Yaskawa INFORM job: MASTER_X2.JBI

/JOB
//NAME MASTER_X2
///FOLDERNAME MASTER_ODWLOK
//POS
///NPOS 138,138,138,0,0,0
///TOOL 0
///POSTYPE PULSE
///PULSE
C00000=2000,-113621,-91819,0,89172,0
C00001=2000,-113621,-91819,0,89172,0
C00002=2000,-99612,-82443,0,53832,0
C00003=2000,-48025,-60869,0,102856,0
C00004=3643,-76224,-106676,19950,71810,76872
C00005=2000,-130321,-133031,0,28968,0
C00006=2000,-109649,-128472,0,44436,0
C00007=2000,-75195,-120874,0,70216,0
C00008=2000,-52226,-115808,0,87402,0
C00009=2000,-87067,-95572,0,78525,0
C00010=2000,-87067,-95572,0,78525,0
C00011=2000,-87067,-95572,0,78525,0
C00012=-12667,-135547,-130714,31270,45596,0
C00013=-12667,-135547,-130714,31270,45596,0
C00014=-12667,-135547,-130714,31270,45596,0
C00015=-7337,-135032,-132177,15524,30149,37578
C00016=-1415,-134459,-133802,-1969,12985,79332
C00017=-1415,-134459,-133802,-1969,12985,79332
C00018=-15972,-110889,-128286,-10965,59905,-43045
C00019=2800,-56338,-97337,-367,83074,232
C00020=2800,-56338,-97337,-367,83074,232
C00021=2000,-92772,-84335,0,66375,0
C00022=2000,-92772,-84335,0,66375,0
C00023=2000,-92772,-84335,0,66375,0
C00024=2000,-92772,-84335,0,66375,0
C00025=2000,-92055,-48789,0,51065,0
C00026=2000,-92055,-48789,0,51065,0
C00027=2000,-92055,-48789,0,51065,0
C00028=2000,-92055,-48789,0,51065,0
C00029=2348,-136985,-121477,16,96092,119
C00030=2348,-136985,-121477,16,96092,119
C00031=2348,-136985,-121477,16,96092,119
C00032=-9622,-119744,-117240,5707,89112,22022
C00033=-39612,-76551,-106625,19964,71626,76894
C00034=-8691,-94790,-119167,5108,91578,19600
C00035=1903,-101039,-123464,18,98414,-30
C00036=1903,-101039,-123464,18,98414,-30
C00037=1903,-101039,-123464,18,98414,-30
C00038=1903,-101039,-123464,18,98414,-30
C00039=-39612,-76551,-106625,19964,71626,76894
C00040=-39612,-76551,-106625,19964,71626,76894
C00041=-39612,-76551,-106625,19964,71626,76894
C00042=-39612,-76551,-106625,19964,71626,76894
C00043=-39612,-76551,-106625,19964,71626,76894
C00044=-39612,-76551,-106625,19964,71626,76894
C00045=-39612,-76551,-106625,19964,71626,76894
C00046=-39612,-76551,-106625,19964,71626,76894
C00047=-39612,-76551,-106625,19964,71626,76894
C00048=-10776,-116726,-133110,1428,79202,268
C00049=-10776,-116726,-133110,1428,79202,268
C00050=-10907,-117335,-90652,-18762,63715,-59495
C00051=-10907,-117335,-90652,-18762,63715,-59495
C00052=-10776,-116726,-133110,1428,79202,268
C00053=-10776,-116726,-133110,1428,79202,268
C00054=-10907,-117335,-90652,-18762,63715,-59495
C00055=2286,-107682,-96534,-81,71711,101
C00056=2286,-107682,-96534,-81,71711,101
C00057=2286,-107682,-96534,-81,71711,101
C00058=2000,-113393,-91320,0,88983,0
C00059=2000,-113393,-91320,0,88983,0
C00060=2000,-113393,-91320,0,88983,0
C00061=2000,-113393,-91320,0,88983,0
C00062=2000,-113393,-91320,0,88983,0
C00063=-39612,-76551,-106625,19964,71626,76894
C00064=-39612,-76551,-106625,19964,71626,76894
C00065=-39612,-76551,-106625,19964,71626,76894
C00066=-39612,-76551,-106625,19964,71626,76894
C00067=-39612,-76551,-106625,19964,71626,76894
C00068=-39612,-76551,-106625,19964,71626,76894
C00069=15474,202180,164610,0,0,38
C00070=15474,202180,164610,0,0,38
C00071=3643,-76224,-106676,19950,71810,76872
C00072=15474,202180,164610,0,0,38
C00073=15474,202180,164610,0,0,38
C00074=15474,202180,164610,0,0,38
C00075=3643,-76224,-106676,19950,71810,76872
C00076=3643,-61024,-22647,36971,32176,65178
C00077=15474,202180,164610,0,0,38
C00078=3643,-76224,-106676,19950,71810,76872
C00079=1588,-95931,-85547,-536,91020,-79
C00080=1588,-95931,-85547,-536,91020,-79
C00081=2000,-138093,-117084,0,0,0
C00082=3643,-76224,-106676,19950,71810,76872
C00083=2000,-138093,-117084,0,0,0
C00084=2000,-138093,-117084,0,0,0
C00085=1941,-102693,-129564,10,101994,-18
C00086=3643,-76224,-106676,19950,71810,76872
C00087=1074,-84890,-111921,820,92639,-133
C00088=1074,-84890,-111921,820,92639,-133
C00089=1999,-107637,-123410,0,80759,1
C00090=3643,-76224,-106676,19950,71810,76872
C00091=2000,17994,-60377,0,102988,0
C00092=2000,-95440,-72516,0,38121,0
C00093=1074,-84890,-111921,820,92639,-133
C00094=3643,-76224,-106676,19950,71810,76872
C00095=421,-73083,-90384,-286,80877,-488
C00096=421,-73083,-90384,-286,80877,-488
C00097=2000,-112988,-119327,0,83158,0
C00098=3643,-76224,-106676,19950,71810,76872
C00099=2000,-112988,-119327,0,83158,0
C00100=2000,-112988,-119327,0,83158,0
C00101=2000,-112988,-119327,0,83158,0
C00102=2000,-112988,-119327,0,83158,0
C00103=2082,-130750,-111396,-32,62200,31
C00104=3643,-76224,-106676,19950,71810,76872
C00105=2082,-130750,-111396,-32,62200,31
C00106=2082,-130750,-111396,-32,62200,31
C00107=1579,-114561,-88072,141,60969,-160
C00108=1579,-114561,-88072,141,60969,-160
C00109=1579,-114561,-88072,141,60969,-160
C00110=3643,-76224,-106676,19950,71810,76872
C00111=-137109,-187493,-133090,6705,82774,-76786
C00112=3643,-76224,-106676,19950,71810,76872
C00113=1579,-114561,-88072,141,60969,-160
C00114=1579,-114561,-88072,141,60969,-160
C00115=2000,-76909,-65168,0,90368,0
C00116=3643,-76224,-106676,19950,71810,76872
C00117=2000,-76909,-65168,0,90368,0
C00118=2000,-76909,-65168,0,90368,0
C00119=3322,-122452,-100913,-73,83322,449
C00120=3643,-76224,-106676,19950,71810,76872
C00121=3322,-122452,-100913,-73,83322,449
C00122=3322,-122452,-100913,-73,83322,449
C00123=3322,-122452,-100913,-73,83322,449
C00124=3322,-122452,-100913,-73,83322,449
C00125=3322,-122452,-100913,-73,83322,449
C00126=2822,-118876,-115474,-188,81202,276
C00127=2000,-115920,-83969,0,54247,0
C00128=2000,-115920,-83969,0,54247,0
C00129=3271,-119374,-120746,-350,28955,423
C00130=3271,-119374,-120746,-350,28955,423
C00131=3271,-119374,-120746,-350,28955,423
C00132=3271,-119374,-120746,-350,28955,423
C00133=3271,-119374,-120746,-350,28955,423
C00134=3270,-119374,-120745,-350,28960,423
C00135=3270,-119374,-120745,-350,28960,423
C00136=3271,-119374,-120746,-350,28955,423
C00137=2000,-113621,-91819,0,89172,0
BC00000=87189,671070,860070
BC00001=87189,689489,1075229
BC00002=0,666204,302418
BC00003=118464,666204,678996
BC00004=199464,674570,1075173
BC00005=200134,698532,1075229
BC00006=160320,689975,1054047
BC00007=93964,675713,1018743
BC00008=49726,666204,995208
BC00009=66580,674291,1075175
BC00010=66580,674291,1075175
BC00011=66580,674291,1075175
BC00012=78393,670967,1075175
BC00013=78393,670967,1075175
BC00014=78393,670967,1075175
BC00015=64389,679433,1075175
BC00016=48829,688840,1075175
BC00017=48829,688840,1075175
BC00018=21214,672831,1075175
BC00019=194082,666204,1075175
BC00020=194082,666204,1075175
BC00021=244954,666204,1064818
BC00022=244954,666204,1063150
BC00023=244954,666204,804590
BC00024=244954,666204,1062399
BC00025=198883,666204,1060496
BC00026=198883,666204,1063896
BC00027=198883,666204,632238
BC00028=198883,666204,632238
BC00029=133260,671337,1075175
BC00030=133260,671337,1075175
BC00031=133260,671337,1075175
BC00032=179494,672257,1075175
BC00033=295325,674563,1075175
BC00034=207960,671388,1071361
BC00035=178026,670300,1070054
BC00036=178026,670300,1070054
BC00037=178026,670300,1070054
BC00038=178026,670300,1070054
BC00039=295325,674563,1075175
BC00040=295325,674563,1075175
BC00041=295325,674563,1075175
BC00042=295325,674563,1075175
BC00043=295325,674563,1075175
BC00044=295325,674563,1075175
BC00045=295325,674563,1075175
BC00046=295325,674563,1075175
BC00047=295325,674563,1075175
BC00048=165820,667836,1075229
BC00049=165820,667836,1075229
BC00050=165820,667836,534036
BC00051=165820,667836,534036
BC00052=165820,667836,1075229
BC00053=165820,667836,1075229
BC00054=165820,667836,534036
BC00055=84306,671503,1075229
BC00056=84306,671503,1075229
BC00057=84306,671503,1075229
BC00058=87189,666204,1075229
BC00059=87189,666204,1075229
BC00060=87189,666204,1075229
BC00061=87189,666204,1075229
BC00062=87189,666204,1075229
BC00063=295325,674563,1075175
BC00064=295325,674563,1075175
BC00065=295325,674563,1075175
BC00066=295325,674563,1075175
BC00067=295325,674563,1075175
BC00068=295325,674563,1075175
BC00069=0,675528,1075229
BC00070=0,675528,1075229
BC00071=199464,674570,1075173
BC00072=0,675528,1075229
BC00073=0,675528,1075229
BC00074=0,675528,1075229
BC00075=199464,674570,1075173
BC00076=199464,674570,909039
BC00077=0,675528,1075229
BC00078=199464,674570,1075173
BC00079=197645,666204,680424
BC00080=197645,666204,680424
BC00081=166720,666220,1057063
BC00082=199464,674570,1075173
BC00083=166720,666220,1057063
BC00084=166720,666220,1057063
BC00085=210618,668760,578653
BC00086=199464,674570,1075173
BC00087=166172,670726,387185
BC00088=166172,670726,1064365
BC00089=108238,670280,1065889
BC00090=199464,674570,1075173
BC00091=32590,674533,986570
BC00092=30861,666204,744559
BC00093=166172,670726,1045420
BC00094=199464,674570,1075173
BC00095=146443,666204,652625
BC00096=146443,666204,652625
BC00097=91901,666204,1075175
BC00098=199464,674570,1075173
BC00099=91901,666204,1075175
BC00100=91901,666204,1075175
BC00101=91901,666204,1075175
BC00102=91901,666204,1075175
BC00103=147868,666204,1075175
BC00104=199464,674570,1075173
BC00105=147868,666204,1075175
BC00106=147868,666204,1075175
BC00107=127053,672594,1075229
BC00108=127053,672594,1075229
BC00109=127053,672594,1075229
BC00110=199464,674570,1075173
BC00111=267033,683758,1057992
BC00112=199464,674570,1075173
BC00113=127053,672594,1075229
BC00114=127053,672594,1075229
BC00115=0,666204,1063572
BC00116=199464,674570,1075173
BC00117=0,666204,619466
BC00118=0,666204,619466
BC00119=87761,666220,1075229
BC00120=199464,674570,1075173
BC00121=87761,666220,1075229
BC00122=87761,666220,1075229
BC00123=87761,666220,1075229
BC00124=87761,666220,1075229
BC00125=87761,666220,1075229
BC00126=0,666204,878766
BC00127=262890,666204,990547
BC00128=262890,666204,990547
BC00129=132383,666204,1075229
BC00130=132383,666204,1075229
BC00131=132383,666204,1075229
BC00132=132383,666204,1075229
BC00133=132383,666204,1075229
BC00134=132383,666204,1075226
BC00135=132383,666204,1075226
BC00136=132383,666204,1075229
BC00137=86234,663735,651575
EC00000=0,0
EC00001=0,0
EC00002=798156,0
EC00003=798156,1112951
EC00004=798156,1112951
EC00005=-798156,1112951
EC00006=-869104,834713
EC00007=-869104,278237
EC00008=-798156,0
EC00009=-798156,1112951
EC00010=-266052,1112951
EC00011=266052,0
EC00012=798156,0
EC00013=798156,0
EC00014=266052,0
EC00015=266052,556475
EC00016=266052,1112951
EC00017=798156,1112951
EC00018=798156,1112951
EC00019=-798156,0
EC00020=-266052,0
EC00021=266052,1112951
EC00022=798156,1112951
EC00023=798156,1112951
EC00024=266052,1112951
EC00025=-5855,0
EC00026=798156,0
EC00027=798156,0
EC00028=266052,0
EC00029=-443420,-556475
EC00030=-798156,-556475
EC00031=-266052,-556475
EC00032=240191,-52511
EC00033=1507629,0
EC00034=1445784,-556475
EC00035=1330261,-556475
EC00036=1330261,-556475
EC00037=1596313,-556475
EC00038=1507629,0
EC00039=-1507629,0
EC00040=-1596313,-556475
EC00041=-1463287,-556475
EC00042=-1463287,-556475
EC00043=-1463287,-556475
EC00044=-1463287,-556475
EC00045=-1596313,-556475
EC00046=-1596313,0
EC00047=-266052,0
EC00048=266052,1112951
EC00049=798156,1112951
EC00050=798156,1112951
EC00051=266052,1112951
EC00052=266052,0
EC00053=798156,0
EC00054=798156,0
EC00055=798156,0
EC00056=798156,0
EC00057=266052,0
EC00058=266052,1112951
EC00059=798156,1112951
EC00060=798156,1112951
EC00061=266052,1112951
EC00062=-266052,0
EC00063=-1507629,0
EC00064=-1596313,-556475
EC00065=-1463287,-556475
EC00066=-1463287,-556475
EC00067=-1596313,-556475
EC00068=-1507629,0
EC00069=-266052,0
EC00070=266052,-556475
EC00071=1108551,-556475
EC00072=-1108551,556475
EC00073=-266052,556475
EC00074=266052,-556475
EC00075=1108551,-556475
EC00076=1108551,-556475
EC00077=-1108551,556475
EC00078=798155,556475
EC00079=798156,556475
EC00080=266052,556475
EC00081=266052,-556475
EC00082=798156,-556475
EC00083=798156,-556475
EC00084=266052,-556475
EC00085=266052,0
EC00086=798156,0
EC00087=798156,0
EC00088=266052,0
EC00089=-266050,1112951
EC00090=-798156,1112951
EC00091=-798156,0
EC00092=-266052,0
EC00093=266052,1112951
EC00094=798156,1112951
EC00095=798156,1112951
EC00096=1596313,1112951
EC00097=1596313,-556475
EC00098=1330261,-556475
EC00099=1330261,-556475
EC00100=1596313,-556475
EC00101=1507629,0
EC00102=266052,0
EC00103=266052,556475
EC00104=780419,556475
EC00105=780419,556475
EC00106=266052,556475
EC00107=-266052,0
EC00108=-798156,0
EC00109=-1585256,0
EC00110=-1527674,557300
EC00111=-1488721,-954
EC00112=-798156,0
EC00113=798156,0
EC00114=266052,0
EC00115=266052,556475
EC00116=798154,556474
EC00117=798156,556475
EC00118=266052,556475
EC00119=266052,1112951
EC00120=798156,1112951
EC00121=798156,1112951
EC00122=266052,1112951
EC00123=266052,0
EC00124=798156,0
EC00125=798156,0
EC00126=1596313,0
EC00127=1596313,-556475
EC00128=1596313,0
EC00129=266052,0
EC00130=266052,556475
EC00131=443420,556475
EC00132=266052,556475
EC00133=0,0
EC00134=-77843,-555115
EC00135=-77843,-555115
EC00136=0,0
EC00137=0,0
//INST
///DATE 2024/12/20 09:57
///ATTR SC,RW
///GROUP1 RB1,BS1
///GROUP2 ST1
NOP
WAIT IG#(285)=255
CLEAR B060 1
'MASTER
SETTM TM000 TRESET
SETTM TM000 TSTART
COMM DOUT OT#(1433) ON
DOUT OT#(1434) ON
MOVJ C00000 BC00000 VJ=100.00  +MOVJ EC00000 VJ=100.00
MOVJ C00001 BC00001 VJ=100.00  +MOVJ EC00001 VJ=100.00
CALL JOB:CLEAN-R1_KM_3P
MOVJ C00002 BC00002 VJ=100.00  +MOVJ EC00002 VJ=100.00
CALL JOB:X2_99(90,0)
MOVJ C00003 BC00003 VJ=100.00  +MOVJ EC00003 VJ=100.00
'
'
MOVJ C00004 BC00004 VJ=100.00  +MOVJ EC00004 VJ=100.00
CALL JOB:CLEAN-R1_KM_NEW
CALL JOB:X2_242(90,180)
MOVJ C00005 BC00005 VJ=100.00  +MOVJ EC00005 VJ=100.00
'
MOVJ C00006 BC00006 VJ=100.00  +MOVJ EC00006 VJ=100.00
MOVJ C00007 BC00007 VJ=100.00  +MOVJ EC00007 VJ=100.00
'
MOVJ C00008 BC00008 VJ=100.00  +MOVJ EC00008 VJ=100.00
CALL JOB:CLEAN-R1_KM_NEW
CALL JOB:X2_6-7(-90,0)
MOVJ C00009 BC00009 VJ=100.00  +MOVJ EC00009 VJ=100.00
'
MOVJ C00010 BC00010 VJ=100.00  +MOVJ EC00010 VJ=100.00
MOVJ C00011 BC00011 VJ=100.00  +MOVJ EC00011 VJ=100.00
'
MOVJ C00012 BC00012 VJ=100.00  +MOVJ EC00012 VJ=100.00
CALL JOB:X2_8A-21A(90,0)
MOVJ C00013 BC00013 VJ=100.00  +MOVJ EC00013 VJ=100.00
'
MOVJ C00014 BC00014 VJ=100.00  +MOVJ EC00014 VJ=100.00
MOVJ C00015 BC00015 VJ=100.00  +MOVJ EC00015 VJ=100.00
MOVJ C00016 BC00016 VJ=100.00  +MOVJ EC00016 VJ=100.00
'
MOVJ C00017 BC00017 VJ=100.00  +MOVJ EC00017 VJ=100.00
CALL JOB:CLEAN-R1_KM_NEW
CALL JOB:X2_8B-21B(90,180)
MOVJ C00018 BC00018 VJ=100.00  +MOVJ EC00018 VJ=100.00
CALL JOB:CLEAN-R1_KM_NEW
'
'
CALL JOB:X2_22-23(-90,180)
MOVJ C00019 BC00019 VJ=100.00  +MOVJ EC00019 VJ=100.00
'
MOVJ C00020 BC00020 VJ=100.00  +MOVJ EC00020 VJ=100.00
MOVJ C00021 BC00021 VJ=100.00  +MOVJ EC00021 VJ=100.00
'
MOVJ C00022 BC00022 VJ=100.00  +MOVJ EC00022 VJ=100.00
CALL JOB:CLEAN-R1_KM_NEW
CALL JOB:X2_24A(90,180)
MOVJ C00023 BC00023 VJ=100.00  +MOVJ EC00023 VJ=100.00
'
MOVJ C00024 BC00024 VJ=100.00  +MOVJ EC00024 VJ=100.00
MOVJ C00025 BC00025 VJ=100.00  +MOVJ EC00025 VJ=100.00
'
MOVJ C00026 BC00026 VJ=100.00  +MOVJ EC00026 VJ=100.00
CALL JOB:CLEAN-R1_KM_NEW
CALL JOB:X2_24B(90,0)
MOVJ C00027 BC00027 VJ=100.00  +MOVJ EC00027 VJ=100.00
'
MOVJ C00028 BC00028 VJ=100.00  +MOVJ EC00028 VJ=100.00
'
MOVJ C00029 BC00029 VJ=100.00  +MOVJ EC00029 VJ=100.00
CALL JOB:CLEAN-R1_KM_NEW
CALL JOB:X2_27-28(-50,-90)
MOVJ C00030 BC00030 VJ=100.00  +MOVJ EC00030 VJ=100.00
'NOWY PRZEJAZD
'
MOVJ C00031 BC00031 VJ=100.00  +MOVJ EC00031 VJ=100.00
MOVJ C00032 BC00032 VJ=100.00  +MOVJ EC00032 VJ=100.00
MOVJ C00033 BC00033 VJ=100.00  +MOVJ EC00033 VJ=100.00
MOVJ C00034 BC00034 VJ=100.00  +MOVJ EC00034 VJ=100.00
'
MOVJ C00035 BC00035 VJ=100.00  +MOVJ EC00035 VJ=100.00
CALL JOB:X2_7,2(150,-90)
MOVJ C00036 BC00036 VJ=100.00  +MOVJ EC00036 VJ=100.00
'
MOVJ C00037 BC00037 VJ=100.00  +MOVJ EC00037 VJ=100.00
MOVJ C00038 BC00038 VJ=100.00  +MOVJ EC00038 VJ=100.00
MOVJ C00039 BC00039 VJ=100.00  +MOVJ EC00039 VJ=100.00
MOVJ C00040 BC00040 VJ=100.00  +MOVJ EC00040 VJ=100.00
'
MOVJ C00041 BC00041 VJ=100.00  +MOVJ EC00041 VJ=100.00
CALL JOB:CLEAN-R1_KM_NEW
CALL JOB:X2_7,1(-165,-90)0
MOVJ C00042 BC00042 VJ=100.00  +MOVJ EC00042 VJ=100.00
'
'
MOVJ C00043 BC00043 VJ=100.00  +MOVJ EC00043 VJ=100.00
CALL JOB:CLEAN-R1_KM_NEW
CALL JOB:X2_34(P)(-165,-90)
MOVJ C00044 BC00044 VJ=100.00  +MOVJ EC00044 VJ=100.00
'
MOVJ C00045 BC00045 VJ=100.00  +MOVJ EC00045 VJ=100.00
MOVJ C00046 BC00046 VJ=100.00  +MOVJ EC00046 VJ=100.00
MOVJ C00047 BC00047 VJ=100.00  +MOVJ EC00047 VJ=100.00
MOVJ C00048 BC00048 VJ=100.00  +MOVJ EC00048 VJ=100.00
'
MOVJ C00049 BC00049 VJ=100.00  +MOVJ EC00049 VJ=100.00
CALL JOB:CLEAN-R1_KM_NEW
CALL JOB:X2_38-47,64(1)(90,180)
MOVJ C00050 BC00050 VJ=100.00  +MOVJ EC00050 VJ=100.00
'
MOVJ C00051 BC00051 VJ=100.00  +MOVJ EC00051 VJ=100.00
MOVJ C00052 BC00052 VJ=100.00  +MOVJ EC00052 VJ=100.00
'
MOVJ C00053 BC00053 VJ=100.00  +MOVJ EC00053 VJ=100.00
CALL JOB:CLEAN-R1_KM_NEW
CALL JOB:X2_38-47,64(2)(90,0)
MOVJ C00054 BC00054 VJ=100.00  +MOVJ EC00054 VJ=100.00
'
'
MOVJ C00055 BC00055 VJ=100.00  +MOVJ EC00055 VJ=100.00
CALL JOB:CLEAN-R1_KM_NEW
CALL JOB:X2_50&56A(90,0)
MOVJ C00056 BC00056 VJ=100.00  +MOVJ EC00056 VJ=100.00
'
MOVJ C00057 BC00057 VJ=100.00  +MOVJ EC00057 VJ=100.00
MOVJ C00058 BC00058 VJ=100.00  +MOVJ EC00058 VJ=100.00
'
MOVJ C00059 BC00059 VJ=100.00  +MOVJ EC00059 VJ=100.00
CALL JOB:CLEAN-R1_KM_NEW
CALL JOB:X2_50&56B(90_180)
MOVJ C00060 BC00060 VJ=100.00  +MOVJ EC00060 VJ=100.00
'
MOVJ C00061 BC00061 VJ=100.00  +MOVJ EC00061 VJ=100.00
MOVJ C00062 BC00062 VJ=100.00  +MOVJ EC00062 VJ=100.00
MOVJ C00063 BC00063 VJ=100.00  +MOVJ EC00063 VJ=100.00
MOVJ C00064 BC00064 VJ=100.00  +MOVJ EC00064 VJ=100.00
'
MOVJ C00065 BC00065 VJ=100.00  +MOVJ EC00065 VJ=100.00
CALL JOB:CLEAN-R1_KM_NEW
CALL JOB:X2_51(P)(-165,-90)
MOVJ C00066 BC00066 VJ=100.00  +MOVJ EC00066 VJ=100.00
'
MOVJ C00067 BC00067 VJ=100.00  +MOVJ EC00067 VJ=100.00
MOVJ C00068 BC00068 VJ=100.00  +MOVJ EC00068 VJ=100.00
MOVJ C00069 BC00069 VJ=100.00  +MOVJ EC00069 VJ=100.00
MOVJ C00070 BC00070 VJ=100.00  +MOVJ EC00070 VJ=100.00
'
MOVJ C00071 BC00071 VJ=100.00  +MOVJ EC00071 VJ=100.00
CALL JOB:CLEAN-R1_KM_NEW
CALL JOB:X2_100(P)(125,-90)
MOVJ C00072 BC00072 VJ=100.00  +MOVJ EC00072 VJ=100.00
'
MOVJ C00073 BC00073 VJ=100.00  +MOVJ EC00073 VJ=100.00
MOVJ C00074 BC00074 VJ=100.00  +MOVJ EC00074 VJ=100.00
'
MOVJ C00075 BC00075 VJ=100.00  +MOVJ EC00075 VJ=100.00
MOVJ C00076 BC00076 VJ=100.00  +MOVJ EC00076 VJ=100.00
PAUSE
'UWAGA!!!!!!!!
'WYMIANA KONCOWKI PRADOWEJ
CALL JOB:CLEAN-R1_KM_NEW
CALL JOB:X2_101(P)(125,-90)2
MOVJ C00077 BC00077 VJ=100.00  +MOVJ EC00077 VJ=100.00
'
'
MOVJ C00078 BC00078 VJ=100.00  +MOVJ EC00078 VJ=100.00
CALL JOB:CLEAN-R1_KM_NEW
CALL JOB:X2_54(90,90)
MOVJ C00079 BC00079 VJ=100.00  +MOVJ EC00079 VJ=100.00
'
MOVJ C00080 BC00080 VJ=100.00  +MOVJ EC00080 VJ=100.00
MOVJ C00081 BC00081 VJ=100.00  +MOVJ EC00081 VJ=100.00
'
MOVJ C00082 BC00082 VJ=100.00  +MOVJ EC00082 VJ=100.00
CALL JOB:CLEAN-R1_KM_NEW
CALL JOB:X2_102(P)(90,-90)1
MOVJ C00083 BC00083 VJ=100.00  +MOVJ EC00083 VJ=100.00
'
MOVJ C00084 BC00084 VJ=100.00  +MOVJ EC00084 VJ=100.00
MOVJ C00085 BC00085 VJ=100.00  +MOVJ EC00085 VJ=100.00
'
MOVJ C00086 BC00086 VJ=100.00  +MOVJ EC00086 VJ=100.00
CALL JOB:CLEAN-R1_KM_NEW
CALL JOB:X2_57-69(1)(90,0)
MOVJ C00087 BC00087 VJ=100.00  +MOVJ EC00087 VJ=100.00
'
MOVJ C00088 BC00088 VJ=100.00  +MOVJ EC00088 VJ=100.00
MOVJ C00089 BC00089 VJ=100.00  +MOVJ EC00089 VJ=100.00
'
MOVJ C00090 BC00090 VJ=100.00  +MOVJ EC00090 VJ=100.00
CALL JOB:CLEAN-R1_KM_NEW
CALL JOB:X2_29-32(-90,180)
MOVJ C00091 BC00091 VJ=100.00  +MOVJ EC00091 VJ=100.00
'
MOVJ C00092 BC00092 VJ=100.00  +MOVJ EC00092 VJ=100.00
MOVJ C00093 BC00093 VJ=100.00  +MOVJ EC00093 VJ=100.00
'
MOVJ C00094 BC00094 VJ=100.00  +MOVJ EC00094 VJ=100.00
CALL JOB:CLEAN-R1_KM_NEW
CALL JOB:X2_57-69(2)(90,180)
MOVJ C00095 BC00095 VJ=100.00  +MOVJ EC00095 VJ=100.00
'
MOVJ C00096 BC00096 VJ=100.00  +MOVJ EC00096 VJ=100.00
MOVJ C00097 BC00097 VJ=100.00  +MOVJ EC00097 VJ=100.00
'
MOVJ C00098 BC00098 VJ=100.00  +MOVJ EC00098 VJ=100.00
CALL JOB:CLEAN-R1_KM_NEW
CALL JOB:X2_48(150,-90)
MOVJ C00099 BC00099 VJ=100.00  +MOVJ EC00099 VJ=100.00
'
MOVJ C00100 BC00100 VJ=100.00  +MOVJ EC00100 VJ=100.00
MOVJ C00101 BC00101 VJ=100.00  +MOVJ EC00101 VJ=100.00
MOVJ C00102 BC00102 VJ=100.00  +MOVJ EC00102 VJ=100.00
MOVJ C00103 BC00103 VJ=100.00  +MOVJ EC00103 VJ=100.00
'
MOVJ C00104 BC00104 VJ=100.00  +MOVJ EC00104 VJ=100.00
CALL JOB:CLEAN-R1_KM_NEW
CALL JOB:X2_49(88,90)
MOVJ C00105 BC00105 VJ=100.00  +MOVJ EC00105 VJ=100.00
'
MOVJ C00106 BC00106 VJ=100.00  +MOVJ EC00106 VJ=100.00
MOVJ C00107 BC00107 VJ=100.00  +MOVJ EC00107 VJ=100.00
'
MOVJ C00108 BC00108 VJ=100.00  +MOVJ EC00108 VJ=100.00
'NOWY PROGRAM NA SCHODKI
MOVJ C00109 BC00109 VJ=100.00  +MOVJ EC00109 VJ=100.00
MOVJ C00110 BC00110 VJ=100.00  +MOVJ EC00110 VJ=100.00
CALL JOB:CLEAN-R1_KM_NEW
CALL JOB:X2_NOWY2
MOVJ C00111 BC00111 VJ=100.00  +MOVJ EC00111 VJ=100.00
MOVJ C00112 BC00112 VJ=100.00  +MOVJ EC00112 VJ=100.00
CALL JOB:CLEAN-R1_KM_NEW
'PROG DO POP
CALL JOB:X2_34-37(-90,0)
MOVJ C00113 BC00113 VJ=100.00  +MOVJ EC00113 VJ=100.00
'
MOVJ C00114 BC00114 VJ=100.00  +MOVJ EC00114 VJ=100.00
MOVJ C00115 BC00115 VJ=100.00  +MOVJ EC00115 VJ=100.00
'
MOVJ C00116 BC00116 VJ=100.00  +MOVJ EC00116 VJ=100.00
CALL JOB:CLEAN-R1_KM_NEW
CALL JOB:X2_25(90,90)
MOVJ C00117 BC00117 VJ=100.00  +MOVJ EC00117 VJ=100.00
'
MOVJ C00118 BC00118 VJ=100.00  +MOVJ EC00118 VJ=100.00
MOVJ C00119 BC00119 VJ=100.00  +MOVJ EC00119 VJ=100.00
'
MOVJ C00120 BC00120 VJ=100.00  +MOVJ EC00120 VJ=100.00
CALL JOB:CLEAN-R1_KM_NEW
CALL JOB:X2_55A(90,180)
MOVJ C00121 BC00121 VJ=100.00  +MOVJ EC00121 VJ=100.00
'
MOVJ C00122 BC00122 VJ=100.00  +MOVJ EC00122 VJ=100.00
MOVJ C00123 BC00123 VJ=100.00  +MOVJ EC00123 VJ=100.00
'
MOVJ C00124 BC00124 VJ=100.00  +MOVJ EC00124 VJ=100.00
CALL JOB:CLEAN-R1_KM_NEW
CALL JOB:X2_55B(90,0)
MOVJ C00125 BC00125 VJ=100.00  +MOVJ EC00125 VJ=100.00
'
'
MOVJ C00126 BC00126 VJ=100.00  +MOVJ EC00126 VJ=100.00
CALL JOB:CLEAN-R1_KM_NEW
CALL JOB:X2_104(180,0)
MOVJ C00127 BC00127 VJ=100.00  +MOVJ EC00127 VJ=100.00
'
MOVJ C00128 BC00128 VJ=100.00  +MOVJ EC00128 VJ=100.00
MOVJ C00129 BC00129 VJ=100.00  +MOVJ EC00129 VJ=100.00
'
MOVJ C00130 BC00130 VJ=100.00  +MOVJ EC00130 VJ=100.00
CALL JOB:CLEAN-R1_KM_NEW
CALL JOB:X2_103(30,90)
MOVJ C00131 BC00131 VJ=100.00  +MOVJ EC00131 VJ=100.00
'
MOVJ C00132 BC00132 VJ=100.00  +MOVJ EC00132 VJ=100.00
MOVJ C00133 BC00133 VJ=100.00  +MOVJ EC00133 VJ=100.00
MOVJ C00134 BC00134 VJ=100.00  +MOVJ EC00134 VJ=100.00
CALL JOB:CLEAN-R1_KM_NEW
CALL JOB:X2_NOWY
COMM DOUT OT#(1433) OFF
DOUT OT#(1434) OFF
MOVJ C00135 BC00135 VJ=100.00  +MOVJ EC00135 VJ=100.00
MOVJ C00136 BC00136 VJ=100.00  +MOVJ EC00136 VJ=100.00
MOVJ C00137 BC00137 VJ=100.00  +MOVJ EC00137 VJ=100.00
SETTM TM000 TSTOP
PAUSE
PAUSE
PAUSE
'
END
